TYPE ST_PuckLockerIO :
STRUCT
	bPuckLockerSensor1		AT %I* : BOOL;
	bPuckLockerSensor2		AT %I* : BOOL;
	bPuckLockerCylinder		AT %Q* : BOOL;
END_STRUCT
END_TYPE

(* stored: Version 1.1.0.1
   DUT ST_PuckLockerIO: Id {48aae017-85d5-4875-a3f2-de429219d00c} *)
